(* IEC 61131-3 sources: tree-sitter-st/tests/std, 11 files *)

(* ---- bistable.st ---- *)
(*
 * An IEC 61131-3 compiler.
 *
 * Based on the
 * FINAL DRAFT - IEC 61131-3, 2nd Ed. (2001-12-10)
 *
 *)

(*
 * This is part of the library conatining the functions
 * and function blocks defined in the standard.
 *
 * SR and RS function blocks
 * -------------------------
 *)

(* The standard defines the SR FB thus:

                  +-----+
S1----------------| >=1 |---Q1
         +---+    |     |
 R------O| & |----|     |
 Q1------|   |    |     |
         +---+    +-----+
*)

FUNCTION_BLOCK SR
  VAR_INPUT
    S1, R : BOOL;
  END_VAR
  VAR_OUTPUT
    Q1 : BOOL;
  END_VAR
  Q1 := S1 OR ((NOT R) AND Q1);
END_FUNCTION_BLOCK

(* The standard defines the RS FB thus:
                   +---+
R1----------------O| & |---Q1
        +-----+    |   |
S-------| >=1 |----|   |
Q1------|     |    |   |
        +-----+    +---+
*)

FUNCTION_BLOCK RS
  VAR_INPUT
    S, R1 : BOOL;
  END_VAR
  VAR_OUTPUT
    Q1 : BOOL;
  END_VAR
  Q1 := (NOT R1) AND (S OR Q1);
END_FUNCTION_BLOCK

(* ---- counter.st ---- *)
(* Following taken directly from the IEC 61131.3 draft standard *)

(*
 * An IEC 61131-3 IL and ST compiler.
 *
 * Based on the
 * FINAL DRAFT - IEC 61131-3, 2nd Ed. (2001-12-10)
 *
 *)

(*
 * This is part of the library conatining the functions
 * and function blocks defined in the standard.
 *
 * Counter function blocks
 * -----------------------
 *)

(******************)
(*                *)
(*    C  T  U     *)
(*                *)
(******************)

FUNCTION_BLOCK CTU
  VAR_INPUT
    CU : BOOL;
    R : BOOL;
    PV : INT;
  END_VAR
  VAR_OUTPUT
    Q : BOOL;
    CV : INT;
  END_VAR
  VAR
    CU_T: R_TRIG;
  END_VAR

  CU_T(CU);
  IF R THEN CV := 0 ;
  ELSIF CU_T.Q AND (CV < PV)
       THEN CV := CV+1;
  END_IF ;
  Q := (CV >= PV) ;
END_FUNCTION_BLOCK

FUNCTION_BLOCK CTU_DINT
  VAR_INPUT
    CU : BOOL;
    R : BOOL;
    PV : DINT;
  END_VAR
  VAR_OUTPUT
    Q : BOOL;
    CV : DINT;
  END_VAR
  VAR
    CU_T: R_TRIG;
  END_VAR

  CU_T(CU);
  IF R THEN CV := 0 ;
  ELSIF CU_T.Q AND (CV < PV)
       THEN CV := CV+1;
  END_IF ;
  Q := (CV >= PV) ;
END_FUNCTION_BLOCK

FUNCTION_BLOCK CTU_LINT
  VAR_INPUT
    CU : BOOL;
    R : BOOL;
    PV : LINT;
  END_VAR
  VAR_OUTPUT
    Q : BOOL;
    CV : LINT;
  END_VAR
  VAR
    CU_T: R_TRIG;
  END_VAR

  CU_T(CU);
  IF R THEN CV := 0 ;
  ELSIF CU_T.Q AND (CV < PV)
       THEN CV := CV+1;
  END_IF ;
  Q := (CV >= PV) ;
END_FUNCTION_BLOCK

FUNCTION_BLOCK CTU_UDINT
  VAR_INPUT
    CU : BOOL;
    R : BOOL;
    PV : UDINT;
  END_VAR
  VAR_OUTPUT
    Q : BOOL;
    CV : UDINT;
  END_VAR
  VAR
    CU_T: R_TRIG;
  END_VAR

  CU_T(CU);
  IF R THEN CV := 0 ;
  ELSIF CU_T.Q AND (CV < PV)
       THEN CV := CV+1;
  END_IF ;
  Q := (CV >= PV) ;
END_FUNCTION_BLOCK

FUNCTION_BLOCK CTU_ULINT
  VAR_INPUT
    CU : BOOL;
    R : BOOL;
    PV : ULINT;
  END_VAR
  VAR_OUTPUT
    Q : BOOL;
    CV : ULINT;
  END_VAR
  VAR
    CU_T: R_TRIG;
  END_VAR

  CU_T(CU);
  IF R THEN CV := 0 ;
  ELSIF CU_T.Q AND (CV < PV)
       THEN CV := CV+1;
  END_IF ;
  Q := (CV >= PV) ;
END_FUNCTION_BLOCK

(******************)
(*                *)
(*    C  T  D     *)
(*                *)
(******************)

FUNCTION_BLOCK CTD
  VAR_INPUT
    CD : BOOL;
    LD : BOOL;
    PV : INT;
  END_VAR
  VAR_OUTPUT
    Q : BOOL;
    CV : INT;
  END_VAR
  VAR
    CD_T: R_TRIG;
  END_VAR

  CD_T(CD);
  IF LD THEN CV := PV ;
  ELSIF CD_T.Q AND (CV > 0)
      THEN CV := CV-1;
  END_IF ;
  Q := (CV <= 0) ;
END_FUNCTION_BLOCK

FUNCTION_BLOCK CTD_DINT
  VAR_INPUT
    CD : BOOL;
    LD : BOOL;
    PV : DINT;
  END_VAR
  VAR_OUTPUT
    Q : BOOL;
    CV : DINT;
  END_VAR
  VAR
    CD_T: R_TRIG;
  END_VAR

  CD_T(CD);
  IF LD THEN CV := PV ;
  ELSIF CD_T.Q AND (CV > 0)
      THEN CV := CV-1;
  END_IF ;
  Q := (CV <= 0) ;
END_FUNCTION_BLOCK

FUNCTION_BLOCK CTD_LINT
  VAR_INPUT
    CD : BOOL;
    LD : BOOL;
    PV : LINT;
  END_VAR
  VAR_OUTPUT
    Q : BOOL;
    CV : LINT;
  END_VAR
  VAR
    CD_T: R_TRIG;
  END_VAR

  CD_T(CD);
  IF LD THEN CV := PV ;
  ELSIF CD_T.Q AND (CV > 0)
      THEN CV := CV-1;
  END_IF ;
  Q := (CV <= 0) ;
END_FUNCTION_BLOCK

FUNCTION_BLOCK CTD_UDINT
  VAR_INPUT
    CD : BOOL;
    LD : BOOL;
    PV : UDINT;
  END_VAR
  VAR_OUTPUT
    Q : BOOL;
    CV : UDINT;
  END_VAR
  VAR
    CD_T: R_TRIG;
  END_VAR

  CD_T(CD);
  IF LD THEN CV := PV ;
  ELSIF CD_T.Q AND (CV > 0)
      THEN CV := CV-1;
  END_IF ;
  Q := (CV <= 0) ;
END_FUNCTION_BLOCK

FUNCTION_BLOCK CTD_ULINT
  VAR_INPUT
    CD : BOOL;
    LD : BOOL;
    PV : ULINT;
  END_VAR
  VAR_OUTPUT
    Q : BOOL;
    CV : ULINT;
  END_VAR
  VAR
    CD_T: R_TRIG;
  END_VAR

  CD_T(CD);
  IF LD THEN CV := PV ;
  ELSIF CD_T.Q AND (CV > 0)
      THEN CV := CV-1;
  END_IF ;
  Q := (CV <= 0) ;
END_FUNCTION_BLOCK

(********************)
(*                  *)
(*    C  T  U D     *)
(*                  *)
(********************)

FUNCTION_BLOCK CTUD
  VAR_INPUT
    CU : BOOL;
    CD : BOOL;
    R  : BOOL;
    LD : BOOL;
    PV : INT;
  END_VAR
  VAR_OUTPUT
    QU : BOOL;
    QD : BOOL;
    CV : INT;
  END_VAR
  VAR
    CD_T: R_TRIG;
    CU_T: R_TRIG;
  END_VAR

  CD_T(CD);
  CU_T(CU);

  IF R THEN CV := 0 ;
  ELSIF LD THEN CV := PV ;
  ELSE
    IF NOT (CU_T.Q AND CD_T.Q) THEN
      IF CU_T.Q AND (CV < PV)
      THEN CV := CV+1;
      ELSIF CD_T.Q AND (CV > 0)
      THEN CV := CV-1;
      END_IF;
    END_IF;
  END_IF ;
  QU := (CV >= PV) ;
  QD := (CV <= 0) ;
END_FUNCTION_BLOCK

FUNCTION_BLOCK CTUD_DINT
  VAR_INPUT
    CU : BOOL;
    CD : BOOL;
    R  : BOOL;
    LD : BOOL;
    PV : DINT;
  END_VAR
  VAR_OUTPUT
    QU : BOOL;
    QD : BOOL;
    CV : DINT;
  END_VAR
  VAR
    CD_T: R_TRIG;
    CU_T: R_TRIG;
  END_VAR

  CD_T(CD);
  CU_T(CU);

  IF R THEN CV := 0 ;
  ELSIF LD THEN CV := PV ;
  ELSE
    IF NOT (CU_T.Q AND CD_T.Q) THEN
      IF CU_T.Q AND (CV < PV)
      THEN CV := CV+1;
      ELSIF CD_T.Q AND (CV > 0)
      THEN CV := CV-1;
      END_IF;
    END_IF;
  END_IF ;
  QU := (CV >= PV) ;
  QD := (CV <= 0) ;
END_FUNCTION_BLOCK

FUNCTION_BLOCK CTUD_LINT
  VAR_INPUT
    CU : BOOL;
    CD : BOOL;
    R  : BOOL;
    LD : BOOL;
    PV : LINT;
  END_VAR
  VAR_OUTPUT
    QU : BOOL;
    QD : BOOL;
    CV : LINT;
  END_VAR
  VAR
    CD_T: R_TRIG;
    CU_T: R_TRIG;
  END_VAR

  CD_T(CD);
  CU_T(CU);

  IF R THEN CV := 0 ;
  ELSIF LD THEN CV := PV ;
  ELSE
    IF NOT (CU_T.Q AND CD_T.Q) THEN
      IF CU_T.Q AND (CV < PV)
      THEN CV := CV+1;
      ELSIF CD_T.Q AND (CV > 0)
      THEN CV := CV-1;
      END_IF;
    END_IF;
  END_IF ;
  QU := (CV >= PV) ;
  QD := (CV <= 0) ;
END_FUNCTION_BLOCK

FUNCTION_BLOCK CTUD_UDINT
  VAR_INPUT
    CU : BOOL;
    CD : BOOL;
    R  : BOOL;
    LD : BOOL;
    PV : UDINT;
  END_VAR
  VAR_OUTPUT
    QU : BOOL;
    QD : BOOL;
    CV : UDINT;
  END_VAR
  VAR
    CD_T: R_TRIG;
    CU_T: R_TRIG;
  END_VAR

  CD_T(CD);
  CU_T(CU);

  IF R THEN CV := 0 ;
  ELSIF LD THEN CV := PV ;
  ELSE
    IF NOT (CU_T.Q AND CD_T.Q) THEN
      IF CU_T.Q AND (CV < PV)
      THEN CV := CV+1;
      ELSIF CD_T.Q AND (CV > 0)
      THEN CV := CV-1;
      END_IF;
    END_IF;
  END_IF ;
  QU := (CV >= PV) ;
  QD := (CV <= 0) ;
END_FUNCTION_BLOCK

FUNCTION_BLOCK CTUD_ULINT
  VAR_INPUT
    CU : BOOL;
    CD : BOOL;
    R  : BOOL;
    LD : BOOL;
    PV : ULINT;
  END_VAR
  VAR_OUTPUT
    QU : BOOL;
    QD : BOOL;
    CV : ULINT;
  END_VAR
  VAR
    CD_T: R_TRIG;
    CU_T: R_TRIG;
  END_VAR

  CD_T(CD);
  CU_T(CU);

  IF R THEN CV := 0 ;
  ELSIF LD THEN CV := PV ;
  ELSE
    IF NOT (CU_T.Q AND CD_T.Q) THEN
      IF CU_T.Q AND (CV < PV)
      THEN CV := CV+1;
      ELSIF CD_T.Q AND (CV > 0)
      THEN CV := CV-1;
      END_IF;
    END_IF;
  END_IF ;
  QU := (CV >= PV) ;
  QD := (CV <= 0) ;
END_FUNCTION_BLOCK

(* ---- derivative.st ---- *)
(* Following taken directly from the IEC 61131.3 draft standard *)

(*
 * An IEC 61131-3 IL and ST compiler.
 *
 * Based on the
 * FINAL DRAFT - IEC 61131-3, 2nd Ed. (2001-12-10)
 *
 *)

 FUNCTION_BLOCK DERIVATIVE
   VAR_INPUT
     RUN : BOOL ;          (* 0 = reset                  *)
     XIN : REAL ;          (* Input to be differentiated *)
     CYCLE : TIME ;        (* Sampling period            *)
   END_VAR
   VAR_OUTPUT
     XOUT : REAL ;         (* Differentiated output      *)
   END_VAR
   VAR X1, X2, X3 : REAL ; END_VAR
   IF RUN THEN
      XOUT := (3.0 * (XIN - X3) + X1 - X2)
              / (10.0 * TIME_TO_REAL(CYCLE)) ;
      X3 := X2 ; X2 := X1 ; X1 := XIN ;
   ELSE XOUT := 0.0; X1 := XIN ; X2 := XIN ; X3 := XIN ;
   END_IF ;
 END_FUNCTION_BLOCK

(* ---- edge_detection.st ---- *)
(* Following taken directly from the IEC 61131.3 draft standard *)

(*
 * An IEC 61131-3 IL and ST compiler.
 *
 * Based on the
 * FINAL DRAFT - IEC 61131-3, 2nd Ed. (2001-12-10)
 *
 *)

(*
 * This is part of the library conatining the functions
 * and function blocks defined in the standard.
 *
 * Edge detection function blocks
 * ------------------------------
 *)

FUNCTION_BLOCK R_TRIG
     VAR_INPUT  CLK: BOOL; END_VAR
     VAR_OUTPUT  Q: BOOL; END_VAR
     VAR M: BOOL; END_VAR
Q := CLK AND NOT M;
M := CLK;
END_FUNCTION_BLOCK

FUNCTION_BLOCK F_TRIG
     VAR_INPUT  CLK: BOOL; END_VAR
     VAR_OUTPUT   Q: BOOL; END_VAR
     VAR M: BOOL; END_VAR
Q := NOT CLK AND NOT M;
M := NOT CLK;
END_FUNCTION_BLOCK

(* ---- hysteresis.st ---- *)
(* Following taken directly from the IEC 61131.3 draft standard *)

(*
 * An IEC 61131-3 IL and ST compiler.
 *
 * Based on the
 * FINAL DRAFT - IEC 61131-3, 2nd Ed. (2001-12-10)
 *
 *)

FUNCTION_BLOCK HYSTERESIS
    (* Boolean hysteresis on difference *)
    (* of REAL inputs, XIN1 - XIN2      *)
  VAR_INPUT XIN1, XIN2, EPS : REAL; END_VAR
  VAR_OUTPUT Q : BOOL := 0; END_VAR
  IF Q THEN IF XIN1 < (XIN2 - EPS) THEN Q := 0; END_IF ;
  ELSIF XIN1 > (XIN2 + EPS) THEN Q := 1 ;
  END_IF ;
END_FUNCTION_BLOCK

(* ---- integral.st ---- *)
(* Following taken directly from the IEC 61131.3 draft standard *)

(*
 * An IEC 61131-3 IL and ST compiler.
 *
 * Based on the
 * FINAL DRAFT - IEC 61131-3, 2nd Ed. (2001-12-10)
 *
 *)

 FUNCTION_BLOCK INTEGRAL
   VAR_INPUT
     RUN : BOOL ;       (* 1 = integrate, 0 = hold *)
     R1 : BOOL ;        (* Overriding reset        *)
     XIN : REAL ;       (* Input variable          *)
     X0  : REAL ;       (* Initial value           *)
     CYCLE : TIME ;     (* Sampling period         *)
   END_VAR
   VAR_OUTPUT
     Q : BOOL ;         (* NOT R1                  *)
     XOUT : REAL ;      (* Integrated output       *)
   END_VAR
   Q := NOT R1 ;
   IF R1 THEN XOUT := X0 ;
   ELSIF RUN THEN XOUT := XOUT + XIN * TIME_TO_REAL(CYCLE);
   END_IF ;
 END_FUNCTION_BLOCK

(* ---- pid.st ---- *)
(* Following taken directly from the IEC 61131.3 draft standard *)

(*
 * An IEC 61131-3 IL and ST compiler.
 *
 * Based on the
 * FINAL DRAFT - IEC 61131-3, 2nd Ed. (2001-12-10)
 *
 *)

 FUNCTION_BLOCK PID
   VAR_INPUT
     AUTO : BOOL ;        (* 0 - manual , 1 - automatic *)
     PV : REAL ;          (* Process variable *)
     SP : REAL ;          (* Set point *)
     X0 : REAL ;          (* Manual output adjustment - *)
                          (* Typically from transfer station *)
     KP : REAL ;          (* Proportionality constant *)
     TR : REAL ;          (* Reset time *)
     TD : REAL ;          (* Derivative time constant *)
     CYCLE : TIME ;       (* Sampling period *)
   END_VAR
   VAR_OUTPUT XOUT : REAL; END_VAR
   VAR ERROR : REAL ;        (* PV - SP *)
       ITERM : INTEGRAL ;    (* FB for integral term  *)
       DTERM : DERIVATIVE ;  (* FB for derivative term *)
   END_VAR
   ERROR := PV - SP ;
   (*** Adjust ITERM so that XOUT := X0 when AUTO = 0 ***)
   ITERM (RUN := AUTO, R1 := NOT AUTO, XIN := ERROR,
          X0 := TR * (X0 - ERROR), CYCLE := CYCLE) ;
   DTERM (RUN := AUTO, XIN := ERROR, CYCLE := CYCLE) ;
   XOUT := KP * (ERROR + ITERM.XOUT/TR + DTERM.XOUT*TD) ;
 END_FUNCTION_BLOCK

(* ---- ramp.st ---- *)
(* Following taken directly from the IEC 61131.3 draft standard *)

(*
 * An IEC 61131-3 IL and ST compiler.
 *
 * Based on the
 * FINAL DRAFT - IEC 61131-3, 2nd Ed. (2001-12-10)
 *
 *)

 FUNCTION_BLOCK RAMP
   VAR_INPUT
     RUN : BOOL ;      (* 0 - track X0, 1 - ramp to/track X1 *)
     X0,X1 : REAL ;
     TR : TIME ;       (* Ramp duration *)
     CYCLE : TIME ;    (* Sampling period *)
   END_VAR
   VAR_OUTPUT
     BUSY : BOOL ; (* BUSY = 1 during ramping period *)
     XOUT : REAL := 0.0 ;
   END_VAR
   VAR XI : REAL ;       (* Initial value *)
       T : TIME := T#0s; (* Elapsed time of ramp *)
   END_VAR
   BUSY := RUN ;
   IF RUN THEN
      IF T >= TR THEN BUSY := 0 ; XOUT := X1 ;
      ELSE XOUT := XI + (X1-XI) * TIME_TO_REAL(T)
                                / TIME_TO_REAL(TR) ;
           T := T + CYCLE ;
      END_IF ;
   ELSE XOUT := X0 ; XI := X0 ; T := t#0s ;
   END_IF ;
 END_FUNCTION_BLOCK

(* ---- rtc.st ---- *)
(****************************************************************

              RTC - Real-time clock

Q is a copy of IN.

When IN = FALSE, CDT is the current date and time as set by the
PLC driver.

When IN changes from FALSE to TRUE, PDT is stored. As long as IN is
TRUE, CDT is equal to PDT + the amount of time since PDT was loaded.

****************************************************************)

FUNCTION_BLOCK RTC
   VAR_INPUT
     IN : BOOL;                  (* 0 - current time, 1 - load time from
PDT *)
     PDT : DT;                   (* Preset datetime *)
   END_VAR
   VAR_OUTPUT
     Q : BOOL := FALSE;          (* Copy of IN *)
     CDT : DT;                   (* Datetime, current or relative to PDT *)
   END_VAR

   VAR
     PREV_IN : BOOL := FALSE;
     OFFSET : TIME;
     CURRENT_TIME : DT;
   END_VAR

   {__SET_VAR(data__->,CURRENT_TIME,,__CURRENT_TIME)}

   IF IN
   THEN
     IF NOT PREV_IN
     THEN
         OFFSET := PDT - CURRENT_TIME;
     END_IF;

     (* PDT + time since PDT was loaded *)
     CDT := CURRENT_TIME + OFFSET;
   ELSE
     CDT := CURRENT_TIME;
   END_IF;

   Q := IN;
   PREV_IN := IN;

END_FUNCTION_BLOCK

(* ---- sema.st ---- *)
(*
 * (c) 2011 Edouard Tisserant
 *
 * Fake semaphore support, for non preemptive implementation.
 *
 *)

FUNCTION_BLOCK SEMA
  VAR_INPUT
    CLAIM : BOOL;
    RELEASE : BOOL;
  END_VAR
  VAR_OUTPUT
    BUSY : BOOL;
  END_VAR
  VAR
    Q_INTERNAL : BOOL;
  END_VAR

  Q_INTERNAL := CLAIM OR ( Q_INTERNAL AND (NOT RELEASE));
  BUSY := Q_INTERNAL;

END_FUNCTION_BLOCK

(* ---- timer.st ---- *)
(*
 * An IEC 61131-3 compiler.
 *
 * Based on the
 * FINAL DRAFT - IEC 61131-3, 2nd Ed. (2001-12-10)
 *
 *)

(*
 * This is part of the library conatining the functions
 * and function blocks defined in the standard.
 *
 * Timer Function Blocks
 * ---------------------
 *
 * NOTE: The timing diagrams in the comments (except the state variable)
 *       were taken from the IEC 61131-3 standard.
 *)

(****************************************************************

                  TP - pulse timing - state machine

            +--------+     ++ ++   +--------+
       IN   |        |     || ||   |        |
          --+        +-----++-++---+        +---------
            t0       t1    t2 t3    t4       t5
            +----+         +----+  +----+
       Q    |    |         |    |  |    |
          --+    +---------+    +--+    +-------------
            t0   t0+PT    t2 t2+PT t4  t4+PT
         PT      +---+          +       +---+
          :     /    |         /|      /    |
       ET :    /     |        / |     /     |
          :   /      |       /  |    /      |
          :  /       |      /   |   /       |
          0-+        +-----+    +--+        +---------
            t0       t1    t2      t4       t5

        2        +---+          +       +---+
STATE   1   +----+   |     +----|  +----+   |
        0 --+        +-----+    +--+        +---------

****************************************************************)

FUNCTION_BLOCK TP
  VAR_INPUT
    IN : BOOL;  (* first input parameter *)
    PT : TIME;  (* second input parameter *)
  END_VAR
  VAR_OUTPUT
    Q : BOOL := FALSE;  (* first output parameter *)
    ET : TIME := T#0s;  (* second output parameter *)
  END_VAR

  VAR
    STATE : SINT := 0;  (* internal state: 0-reset, 1-counting, 2-set *)
    PREV_IN : BOOL := FALSE;
    CURRENT_TIME, START_TIME : TIME;
  END_VAR

  {__SET_VAR(data__->,CURRENT_TIME,,__CURRENT_TIME)}

  IF ((STATE = 0) AND NOT(PREV_IN) AND IN)   (* found rising edge on IN *)
  THEN
    (* start timer... *)
    STATE := 1;
    Q := TRUE;
    START_TIME := CURRENT_TIME;

  ELSIF (STATE = 1)
  THEN
    IF ((START_TIME + PT) <= CURRENT_TIME)
    THEN
      STATE := 2;
      Q := FALSE;
      ET := PT;
    ELSE
      ET := CURRENT_TIME - START_TIME;
    END_IF;
  END_IF;

  IF ((STATE = 2) AND NOT(IN))
  THEN
    ET := T#0s;
    STATE := 0;
  END_IF;

  PREV_IN := IN;

END_FUNCTION_BLOCK

(****************************************************************

             TON - On-delay timing - state machine

            +--------+        +---+   +--------+
       IN   |        |        |   |   |        |
          --+        +--------+   +---+        +-------------
            t0       t1       t2  t3  t4       t5
                 +---+                     +---+
       Q         |   |                     |   |
          -------+   +---------------------+   +-------------
              t0+PT  t1                t4+PT   t5
         PT      +---+                     +---+
          :     /    |            +       /    |
       ET :    /     |           /|      /     |
          :   /      |          / |     /      |
          :  /       |         /  |    /       |
          0-+        +--------+   +---+        +-------------
            t0       t1       t2  t3  t4       t5

        2        +---+                     +---+
STATE   1   +----+   |        +---+   +----+   |
        0 --+        +--------+   +---+        +------

****************************************************************)

FUNCTION_BLOCK TON
  VAR_INPUT
    IN : BOOL;  (* first input parameter *)
    PT : TIME;  (* second input parameter *)
  END_VAR
  VAR_OUTPUT
    Q : BOOL := FALSE;  (* first output parameter *)
    ET : TIME := T#0s;  (* second output parameter *)
  END_VAR

  VAR
    STATE : SINT := 0;  (* internal state: 0-reset, 1-counting, 2-set *)
    PREV_IN : BOOL := FALSE;
    CURRENT_TIME, START_TIME : TIME;
  END_VAR

  {__SET_VAR(data__->,CURRENT_TIME,,__CURRENT_TIME)}

  IF ((STATE = 0) AND NOT(PREV_IN) AND IN)   (* found rising edge on IN *)
  THEN
    (* start timer... *)
    STATE := 1;
    Q := FALSE;
    START_TIME := CURRENT_TIME;

  ELSE
    (* STATE is 1 or 2 !! *)
    IF (NOT(IN))
    THEN
      ET := T#0s;
      Q := FALSE;
      STATE := 0;

    ELSIF (STATE = 1)
    THEN
      IF ((START_TIME + PT) <= CURRENT_TIME)
      THEN
        STATE := 2;
        Q := TRUE;
        ET := PT;
      ELSE
        ET := CURRENT_TIME - START_TIME;
      END_IF;
    END_IF;

  END_IF;

  PREV_IN := IN;

END_FUNCTION_BLOCK

(****************************************************************

             TOF - Off-delay timing - state machine

              +--------+        +---+   +--------+
       IN     |        |        |   |   |        |
           ---+        +--------+   +---+        +-----------
              t0       t1       t2  t3  t4       t5
              +-------------+   +---------------------+
       Q      |             |   |                     |
           ---+             +---+                     +------
              t0          t1+PT t2                  t5+PT
         PT                 +---+                     +------
          :                /    |       +            /
       ET :               /     |      /|           /
          :              /      |     / |          /
          :             /       |    /  |         /
          0------------+        +---+   +--------+
                       t1           t3           t5

        2                   +---+                     +------
STATE   1              +----+   |   +---+        +----+
        0 -------------+        +---+   +--------+

****************************************************************)

FUNCTION_BLOCK TOF
  VAR_INPUT
    IN : BOOL;  (* first input parameter *)
    PT : TIME;  (* second input parameter *)
  END_VAR
  VAR_OUTPUT
    Q : BOOL := FALSE;  (* first output parameter *)
    ET : TIME := T#0s;  (* second output parameter *)
  END_VAR

  VAR
    STATE : SINT := 0;  (* internal state: 0-reset, 1-counting, 2-set *)
    PREV_IN : BOOL := FALSE;
    CURRENT_TIME, START_TIME : TIME;
  END_VAR

  {__SET_VAR(data__->,CURRENT_TIME,,__CURRENT_TIME)}

  IF ((STATE = 0) AND PREV_IN AND NOT(IN))   (* found falling edge on IN *)
  THEN
    (* start timer... *)
    STATE := 1;
    START_TIME := CURRENT_TIME;

  ELSE
    (* STATE is 1 or 2 !! *)
    IF (IN)
    THEN
      ET := T#0s;
      STATE := 0;

    ELSIF (STATE = 1)
    THEN
      IF ((START_TIME + PT) <= CURRENT_TIME)
      THEN
        STATE := 2;
        ET := PT;
      ELSE
        ET := CURRENT_TIME - START_TIME;
      END_IF;
    END_IF;

  END_IF;

  Q := IN OR (STATE = 1);
  PREV_IN := IN;

END_FUNCTION_BLOCK
